// TIA Portal V19 export
TYPE "typeAxisControlProduction"
// stored: Access Published
   STRUCT
      upperVel : LReal := 100.0;   // 产品模式速度上限
      vel : LReal := 20.0;   // 产品模式设定值，画面做限制根据上限值如果超了不允许输入
      distance1 : LReal := 10.0;   // 产品模式下拉带走的定长距离
      distance2 : LReal;   // 预留
      distanceList : Array[0..199] of "typePosAxisParameter";
      acc : LReal := 0.5;
      dec : LReal := 0.5;
   END_STRUCT;
END_TYPE
